FUNCTION_BLOCK FB_Pulse
VAR_INPUT
	bEnable : BOOL;
	tTimeOn : TIME;
	tTimeOff : TIME;
END_VAR
VAR_OUTPUT
	bPulse : BOOL;
END_VAR
VAR
	tmr1 : TON;
	tmr2 : TOF;
	IN: INT;
END_VAR

tmr1(IN:= bEnable AND NOT tmr2.Q, PT:= tTimeOff, Q=> , ET=> );
tmr2(IN:= tmr1.Q, PT:= tTimeOn, Q=> bPulse, ET=> );

END_FUNCTION_BLOCK

(* stored: Version 1.1.0.1, ProductVersion 3.1.4024.9
   POU FB_Pulse: Id {c3d102ed-a867-4056-8c17-54ee32287f51}, SpecialFunc None *)
